(* Logix 5000 project; controller NSH_PLC2 vendor 1 type 14 code 167 rev 32.14; software revision 32.03; part 2 of 6 *)
(* tags used below, declared in another part *)
   AOI_MCC2_10A_ToPLC1 : E300ToMotor;
   AOI_MCC2_10C_ToPLC1 : E300ToMotor;
   AOI_MCC2_10E_ToPLC1 : E300ToMotor;
   AOI_MCC2_10G_ToPLC1 : E300ToMotor;
   AOI_MCC2_10J_ToPLC1 : E300ToMotor;
   AOI_MCC2_10L_ToPLC1 : E300ToMotor;
   AOI_MCC2_11A_ToPLC1 : E300ToMotor;
   AOI_MCC2_11C_ToPLC1 : E300ToMotor;
   AOI_MCC2_11E_ToPLC1 : E300ToMotor;
   AOI_MCC2_11G_ToPLC1 : E300ToMotor;
   AOI_MCC2_11J_ToPLC1 : E300ToMotor;
   AOI_MCC2_11L_ToPLC1 : E300ToMotor;
   AOI_MCC2_12A_ToPLC1 : E300ToMotor;
   AOI_MCC2_12C_ToPLC1 : E300ToMotor;
   AOI_MCC2_12E_ToPLC1 : E300ToMotor;
   AOI_MCC2_12G_ToPLC1 : E300ToMotor;
   AOI_MCC2_12J_ToPLC1 : E300ToMotor;
   AOI_MCC2_12L_ToPLC1 : E300ToMotor;
   AOI_MCC2_13A_ToPLC1 : E300ToMotor;
   AOI_MCC2_13C_ToPLC1 : E300ToMotor;
   AOI_MCC2_13E_ToPLC1 : E300ToMotor;
   AOI_MCC2_13G_ToPLC1 : E300ToMotor;
   AOI_MCC2_13J_ToPLC1 : E300ToMotor;
   AOI_MCC2_14A_ToPLC1 : E300ToMotor;
   AOI_MCC2_14C_ToPLC1 : E300ToMotor;
   AOI_MCC2_14E_ToPLC1 : E300ToMotor;
   AOI_MCC2_14G_ToPLC1 : E300ToMotor;
   AOI_MCC2_14J_ToPLC1 : E300ToMotor;
   AOI_MCC2_14L_ToPLC1 : E300ToMotor;
   AOI_MCC2_15A_ToPLC1 : E300ToMotor;
   AOI_MCC2_15C_ToPLC1 : E300ToMotor;
   AOI_MCC2_15E_ToPLC1 : E300ToMotor;
   AOI_MCC2_15G_ToPLC1 : E300ToMotor;
   AOI_MCC2_2A_ToPLC1 : PF525ToMotor;
   AOI_MCC2_2D_ToPLC1 : PF525ToMotor;
   AOI_MCC2_2G_ToPLC1 : PF525ToMotor;
   AOI_MCC2_2K_ToPLC1 : PF525ToMotor;
   AOI_MCC2_3A_ToPLC1 : E300ToMotor;
   AOI_MCC2_3C_ToPLC1 : E300ToMotor;
   AOI_MCC2_3E_ToPLC1 : E300ToMotor;
   AOI_MCC2_3G_ToPLC1 : E300ToMotor;
   AOI_MCC2_3J_ToPLC1 : E300ToMotor;
   AOI_MCC2_3L_ToPLC1 : E300ToMotor;
   AOI_MCC2_4A_ToPLC1 : E300ToMotor;
   AOI_MCC2_4C_ToPLC1 : E300ToMotor;
   AOI_MCC2_4E_ToPLC1 : E300ToMotor;
   AOI_MCC2_4G_ToPLC1 : E300ToMotor;
   AOI_MCC2_4J_ToPLC1 : E300ToMotor;
   AOI_MCC2_4L_ToPLC1 : E300ToMotor;
   AOI_MCC2_5A_ToPLC1 : E300ToMotor;
   AOI_MCC2_5C_ToPLC1 : E300ToMotor;
   AOI_MCC2_5E_ToPLC1 : E300ToMotor;
   AOI_MCC2_5G_ToPLC1 : E300ToMotor;
   AOI_MCC2_5J_ToPLC1 : E300ToMotor;
   AOI_MCC2_6A_ToPLC1 : E300ToMotor;
   AOI_MCC2_6C_ToPLC1 : E300ToMotor;
   AOI_MCC2_6E_ToPLC1 : E300ToMotor;
   AOI_MCC2_6G_ToPLC1 : E300ToMotor;
   AOI_MCC2_6J_ToPLC1 : E300ToMotor;
   AOI_MCC2_6L_ToPLC1 : E300ToMotor;
   AOI_MCC2_7A_ToPLC1 : E300ToMotor;
   AOI_MCC2_7D_ToPLC1 : E300ToMotor;
   AOI_MCC2_7G_ToPLC1 : E300ToMotor;
   AOI_MCC2_7K_ToPLC1 : E300ToMotor;
   AOI_MCC2_8B_ToPLC1 : E300ToMotor;
   AOI_MCC2_8D_ToPLC1 : E300ToMotor;
   AOI_MCC2_8F_ToPLC1 : E300ToMotor;
   AOI_MCC2_8H_ToPLC1 : E300ToMotor;
   AOI_MCC2_8K_ToPLC1 : E300ToMotor;
   AOI_MCC2_9D_ToPLC1 : E300ToMotor;
   AOI_MCC2_9F_ToPLC1 : E300ToMotor;
   AOI_MCC2_9H_ToPLC1 : PF525ToMotor;
   Const_4000_Hex : INT;   // Constant #16:4000, Entry Status Communicating
   GSV_EntryStatus : INT;   // GSV Entry Status, shold be #16:4000
   MCC2_10A_CommsOK : BOOL;   // Communications with AOP OK
   MCC2_10C_CommsOK : BOOL;   // Communications with AOP OK
   MCC2_10E_CommsOK : BOOL;   // Communications with AOP OK
   MCC2_10G_CommsOK : BOOL;   // Communications with AOP OK
   MCC2_10J_CommsOK : BOOL;   // Communications with AOP OK
   MCC2_10L_CommsOK : BOOL;   // Communications with AOP OK
   MCC2_11A_CommsOK : BOOL;   // Communications with AOP OK
   MCC2_11C_CommsOK : BOOL;   // Communications with AOP OK
   MCC2_11E_CommsOK : BOOL;   // Communications with AOP OK
   MCC2_11G_CommsOK : BOOL;   // Communications with AOP OK
   MCC2_11J_CommsOK : BOOL;   // Communications with AOP OK
   MCC2_11L_CommsOK : BOOL;   // Communications with AOP OK
   MCC2_12A_CommsOK : BOOL;   // Communications with AOP OK
   MCC2_12C_CommsOK : BOOL;   // Communications with AOP OK
   MCC2_12E_CommsOK : BOOL;   // Communications with AOP OK
   MCC2_12G_CommsOK : BOOL;   // Communications with AOP OK
   MCC2_12J_CommsOK : BOOL;   // Communications with AOP OK
   MCC2_12L_CommsOK : BOOL;   // Communications with AOP OK
   MCC2_13A_CommsOK : BOOL;   // Communications with AOP OK
   MCC2_13C_CommsOK : BOOL;   // Communications with AOP OK
   MCC2_13E_CommsOK : BOOL;   // Communications with AOP OK
   MCC2_13G_CommsOK : BOOL;   // Communications with AOP OK
   MCC2_13J_CommsOK : BOOL;   // Communications with AOP OK
   MCC2_14A_CommsOK : BOOL;   // Communications with AOP OK
   MCC2_14C_CommsOK : BOOL;   // Communications with AOP OK
   MCC2_14E_CommsOK : BOOL;   // Communications with AOP OK
   MCC2_14G_CommsOK : BOOL;   // Communications with AOP OK
   MCC2_14J_CommsOK : BOOL;   // Communications with AOP OK
   MCC2_14L_CommsOK : BOOL;   // Communications with AOP OK
   MCC2_15A_CommsOK : BOOL;   // Communications with AOP OK
   MCC2_15C_CommsOK : BOOL;   // Communications with AOP OK
   MCC2_15E_CommsOK : BOOL;   // Communications with AOP OK
   MCC2_15G_CommsOK : BOOL;   // Communications with AOP OK
   MCC2_2A_CommsOK : BOOL;   // Communications with AOP OK
   MCC2_2D_CommsOK : BOOL;   // Communications with AOP OK
   MCC2_2G_CommsOK : BOOL;   // Communications with AOP OK
   MCC2_2K_CommsOK : BOOL;   // Communications with AOP OK
   MCC2_3A_CommsOK : BOOL;   // Communications with AOP OK
   MCC2_3C_CommsOK : BOOL;   // Communications with AOP OK
   MCC2_3E_CommsOK : BOOL;   // Communications with AOP OK
   MCC2_3G_CommsOK : BOOL;   // Communications with AOP OK
   MCC2_3J_CommsOK : BOOL;   // Communications with AOP OK
   MCC2_3L_CommsOK : BOOL;   // Communications with AOP OK
   MCC2_4A_CommsOK : BOOL;   // Communications with AOP OK
   MCC2_4C_CommsOK : BOOL;   // Communications with AOP OK
   MCC2_4E_CommsOK : BOOL;   // Communications with AOP OK
   MCC2_4G_CommsOK : BOOL;   // Communications with AOP OK
   MCC2_4J_CommsOK : BOOL;   // Communications with AOP OK
   MCC2_4L_CommsOK : BOOL;   // Communications with AOP OK
   MCC2_5A_CommsOK : BOOL;   // Communications with AOP OK
   MCC2_5C_CommsOK : BOOL;   // Communications with AOP OK
   MCC2_5E_CommsOK : BOOL;   // Communications with AOP OK
   MCC2_5G_CommsOK : BOOL;   // Communications with AOP OK
   MCC2_5J_CommsOK : BOOL;   // Communications with AOP OK
   MCC2_6A_CommsOK : BOOL;   // Communications with AOP OK
   MCC2_6C_CommsOK : BOOL;   // Communications with AOP OK
   MCC2_6E_CommsOK : BOOL;   // Communications with AOP OK
   MCC2_6G_CommsOK : BOOL;   // Communications with AOP OK
   MCC2_6J_CommsOK : BOOL;   // Communications with AOP OK
   MCC2_6L_CommsOK1 : BOOL;   // Communications with AOP OK
   MCC2_7A_CommsOK : BOOL;   // Communications with AOP OK
   MCC2_7D_CommsOK : BOOL;   // Communications with AOP OK
   MCC2_7G_CommsOK : BOOL;   // Communications with AOP OK
   MCC2_7K_CommsOK : BOOL;   // Communications with AOP OK
   MCC2_8B_CommsOK : BOOL;   // Communications with AOP OK
   MCC2_8D_CommsOK : BOOL;   // Communications with AOP OK
   MCC2_8F_CommsOK : BOOL;   // Communications with AOP OK
   MCC2_8H_CommsOK : BOOL;   // Communications with AOP OK
   MCC2_8K_CommsOK : BOOL;   // Communications with AOP OK
   MCC2_9D_CommsOK : BOOL;   // Communications with AOP OK
   MCC2_9F_CommsOK : BOOL;   // Communications with AOP OK
   MCC2_9H_CommsOK : BOOL;   // Communications with AOP OK
   MotorsStatusTag : MotorsStatusUDT;   // Only Instance of UDT

PROGRAM MainProgram   (* main routine MainRoutine *)

ROUTINE AOP_ToPLC1   (* ladder *)
// Get Motor AOPs To AllMotorsToPLC1
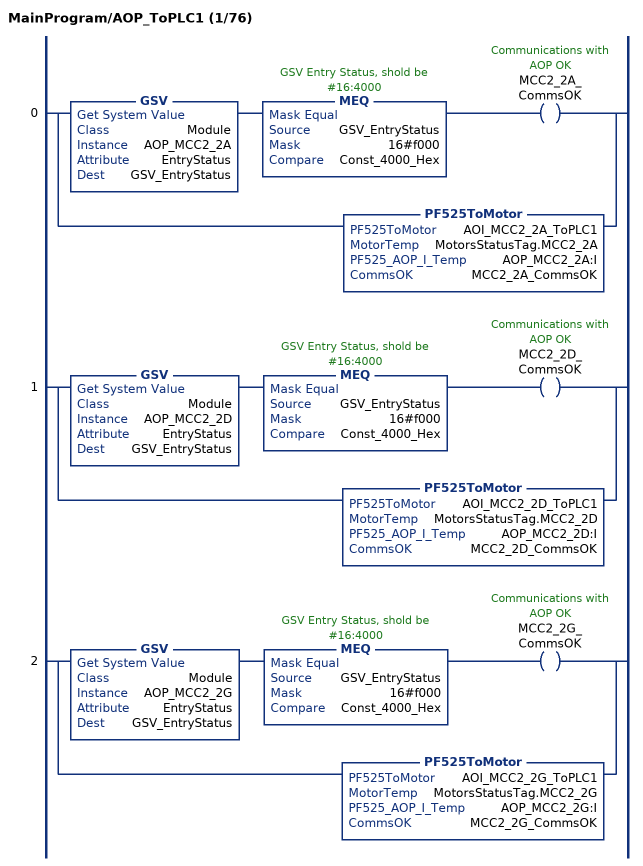
   0: [GSV(Module,AOP_MCC2_2A,EntryStatus,GSV_EntryStatus) MEQ(GSV_EntryStatus,16#f000,Const_4000_Hex) OTE(MCC2_2A_CommsOK) ,PF525ToMotor(AOI_MCC2_2A_ToPLC1,MotorsStatusTag.MCC2_2A,AOP_MCC2_2A:I,MCC2_2A_CommsOK) ];
   1: [GSV(Module,AOP_MCC2_2D,EntryStatus,GSV_EntryStatus) MEQ(GSV_EntryStatus,16#f000,Const_4000_Hex) OTE(MCC2_2D_CommsOK) ,PF525ToMotor(AOI_MCC2_2D_ToPLC1,MotorsStatusTag.MCC2_2D,AOP_MCC2_2D:I,MCC2_2D_CommsOK) ];
   2: [GSV(Module,AOP_MCC2_2G,EntryStatus,GSV_EntryStatus) MEQ(GSV_EntryStatus,16#f000,Const_4000_Hex) OTE(MCC2_2G_CommsOK) ,PF525ToMotor(AOI_MCC2_2G_ToPLC1,MotorsStatusTag.MCC2_2G,AOP_MCC2_2G:I,MCC2_2G_CommsOK) ];
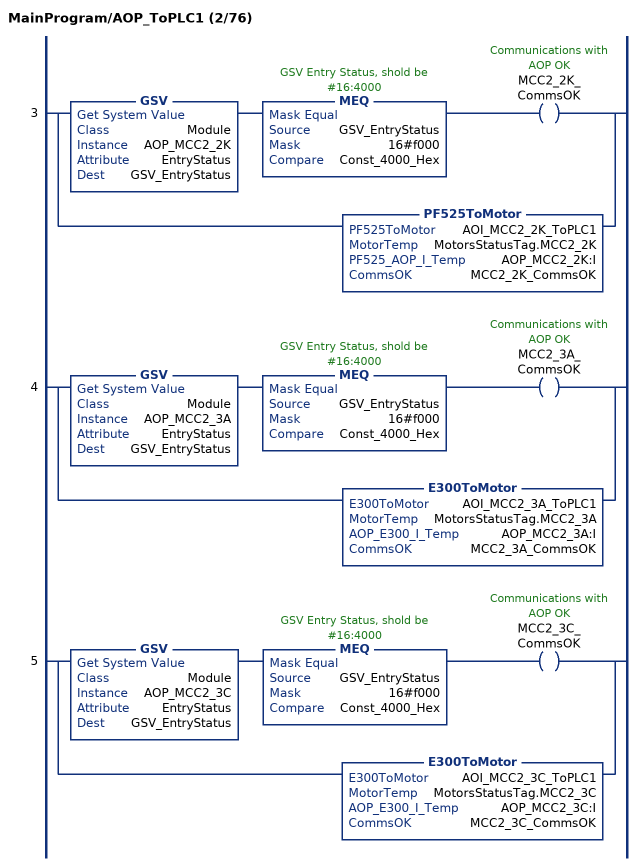
   3: [GSV(Module,AOP_MCC2_2K,EntryStatus,GSV_EntryStatus) MEQ(GSV_EntryStatus,16#f000,Const_4000_Hex) OTE(MCC2_2K_CommsOK) ,PF525ToMotor(AOI_MCC2_2K_ToPLC1,MotorsStatusTag.MCC2_2K,AOP_MCC2_2K:I,MCC2_2K_CommsOK) ];
   4: [GSV(Module,AOP_MCC2_3A,EntryStatus,GSV_EntryStatus) MEQ(GSV_EntryStatus,16#f000,Const_4000_Hex) OTE(MCC2_3A_CommsOK) ,E300ToMotor(AOI_MCC2_3A_ToPLC1,MotorsStatusTag.MCC2_3A,AOP_MCC2_3A:I,MCC2_3A_CommsOK) ];
   5: [GSV(Module,AOP_MCC2_3C,EntryStatus,GSV_EntryStatus) MEQ(GSV_EntryStatus,16#f000,Const_4000_Hex) OTE(MCC2_3C_CommsOK) ,E300ToMotor(AOI_MCC2_3C_ToPLC1,MotorsStatusTag.MCC2_3C,AOP_MCC2_3C:I,MCC2_3C_CommsOK) ];
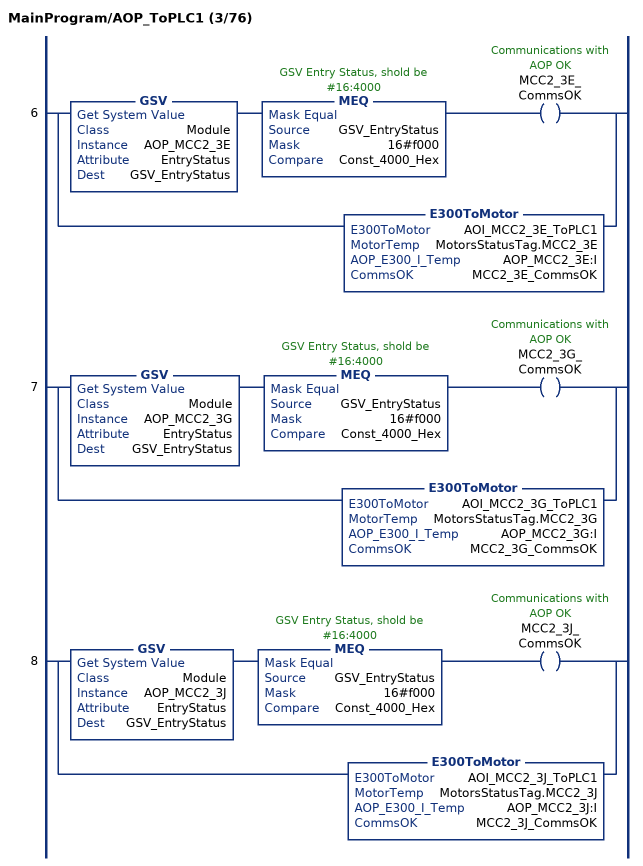
   6: [GSV(Module,AOP_MCC2_3E,EntryStatus,GSV_EntryStatus) MEQ(GSV_EntryStatus,16#f000,Const_4000_Hex) OTE(MCC2_3E_CommsOK) ,E300ToMotor(AOI_MCC2_3E_ToPLC1,MotorsStatusTag.MCC2_3E,AOP_MCC2_3E:I,MCC2_3E_CommsOK) ];
   7: [GSV(Module,AOP_MCC2_3G,EntryStatus,GSV_EntryStatus) MEQ(GSV_EntryStatus,16#f000,Const_4000_Hex) OTE(MCC2_3G_CommsOK) ,E300ToMotor(AOI_MCC2_3G_ToPLC1,MotorsStatusTag.MCC2_3G,AOP_MCC2_3G:I,MCC2_3G_CommsOK) ];
   8: [GSV(Module,AOP_MCC2_3J,EntryStatus,GSV_EntryStatus) MEQ(GSV_EntryStatus,16#f000,Const_4000_Hex) OTE(MCC2_3J_CommsOK) ,E300ToMotor(AOI_MCC2_3J_ToPLC1,MotorsStatusTag.MCC2_3J,AOP_MCC2_3J:I,MCC2_3J_CommsOK) ];
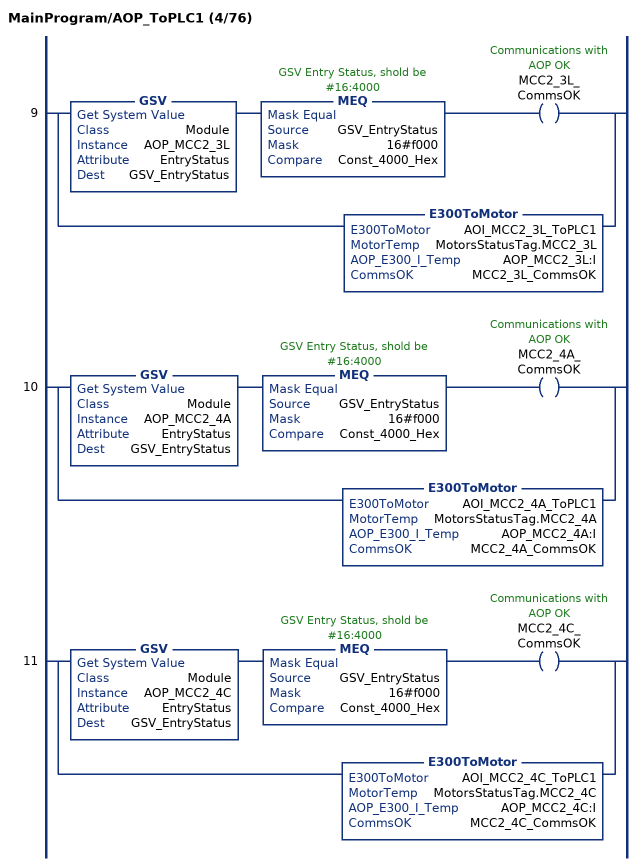
   9: [GSV(Module,AOP_MCC2_3L,EntryStatus,GSV_EntryStatus) MEQ(GSV_EntryStatus,16#f000,Const_4000_Hex) OTE(MCC2_3L_CommsOK) ,E300ToMotor(AOI_MCC2_3L_ToPLC1,MotorsStatusTag.MCC2_3L,AOP_MCC2_3L:I,MCC2_3L_CommsOK) ];
   10: [GSV(Module,AOP_MCC2_4A,EntryStatus,GSV_EntryStatus) MEQ(GSV_EntryStatus,16#f000,Const_4000_Hex) OTE(MCC2_4A_CommsOK) ,E300ToMotor(AOI_MCC2_4A_ToPLC1,MotorsStatusTag.MCC2_4A,AOP_MCC2_4A:I,MCC2_4A_CommsOK) ];
   11: [GSV(Module,AOP_MCC2_4C,EntryStatus,GSV_EntryStatus) MEQ(GSV_EntryStatus,16#f000,Const_4000_Hex) OTE(MCC2_4C_CommsOK) ,E300ToMotor(AOI_MCC2_4C_ToPLC1,MotorsStatusTag.MCC2_4C,AOP_MCC2_4C:I,MCC2_4C_CommsOK) ];
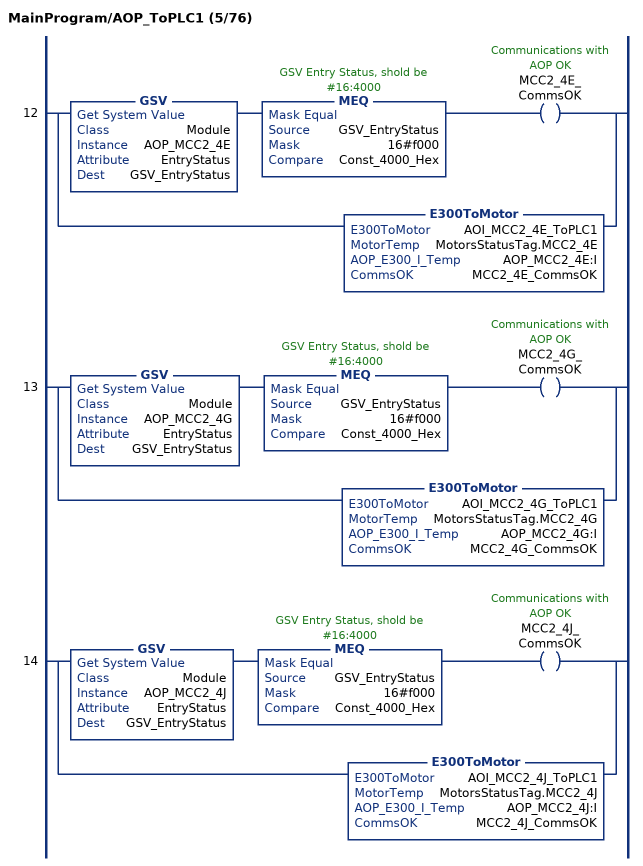
   12: [GSV(Module,AOP_MCC2_4E,EntryStatus,GSV_EntryStatus) MEQ(GSV_EntryStatus,16#f000,Const_4000_Hex) OTE(MCC2_4E_CommsOK) ,E300ToMotor(AOI_MCC2_4E_ToPLC1,MotorsStatusTag.MCC2_4E,AOP_MCC2_4E:I,MCC2_4E_CommsOK) ];
   13: [GSV(Module,AOP_MCC2_4G,EntryStatus,GSV_EntryStatus) MEQ(GSV_EntryStatus,16#f000,Const_4000_Hex) OTE(MCC2_4G_CommsOK) ,E300ToMotor(AOI_MCC2_4G_ToPLC1,MotorsStatusTag.MCC2_4G,AOP_MCC2_4G:I,MCC2_4G_CommsOK) ];
   14: [GSV(Module,AOP_MCC2_4J,EntryStatus,GSV_EntryStatus) MEQ(GSV_EntryStatus,16#f000,Const_4000_Hex) OTE(MCC2_4J_CommsOK) ,E300ToMotor(AOI_MCC2_4J_ToPLC1,MotorsStatusTag.MCC2_4J,AOP_MCC2_4J:I,MCC2_4J_CommsOK) ];
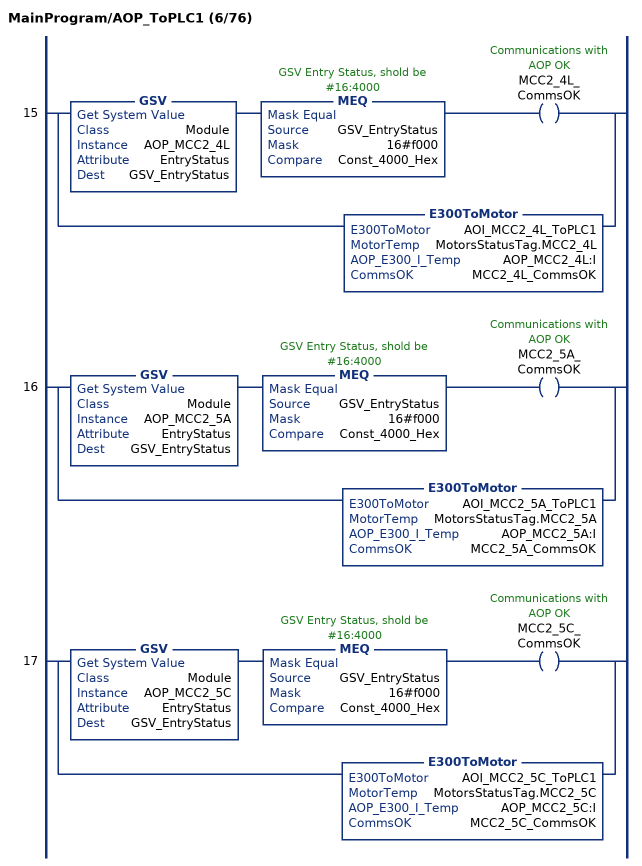
   15: [GSV(Module,AOP_MCC2_4L,EntryStatus,GSV_EntryStatus) MEQ(GSV_EntryStatus,16#f000,Const_4000_Hex) OTE(MCC2_4L_CommsOK) ,E300ToMotor(AOI_MCC2_4L_ToPLC1,MotorsStatusTag.MCC2_4L,AOP_MCC2_4L:I,MCC2_4L_CommsOK) ];
   16: [GSV(Module,AOP_MCC2_5A,EntryStatus,GSV_EntryStatus) MEQ(GSV_EntryStatus,16#f000,Const_4000_Hex) OTE(MCC2_5A_CommsOK) ,E300ToMotor(AOI_MCC2_5A_ToPLC1,MotorsStatusTag.MCC2_5A,AOP_MCC2_5A:I,MCC2_5A_CommsOK) ];
   17: [GSV(Module,AOP_MCC2_5C,EntryStatus,GSV_EntryStatus) MEQ(GSV_EntryStatus,16#f000,Const_4000_Hex) OTE(MCC2_5C_CommsOK) ,E300ToMotor(AOI_MCC2_5C_ToPLC1,MotorsStatusTag.MCC2_5C,AOP_MCC2_5C:I,MCC2_5C_CommsOK) ];
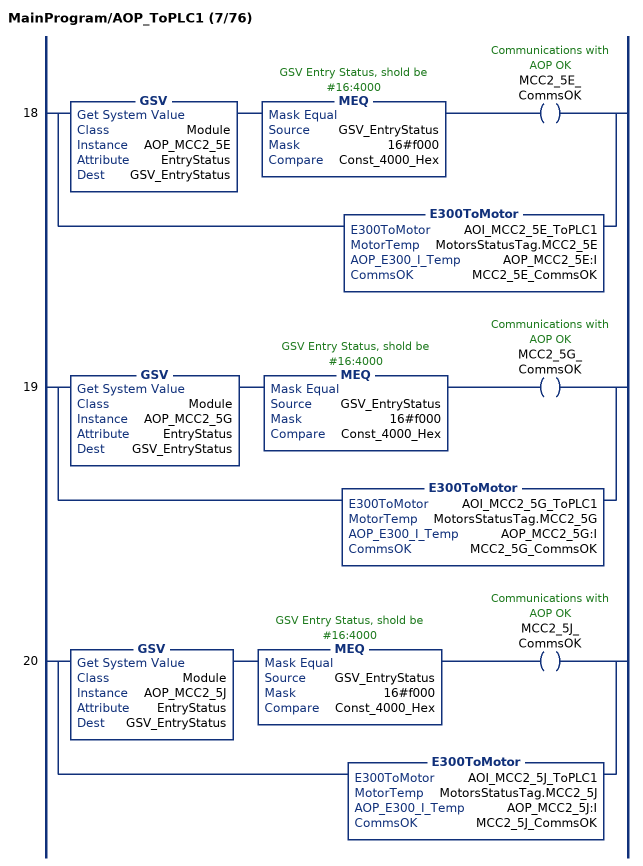
   18: [GSV(Module,AOP_MCC2_5E,EntryStatus,GSV_EntryStatus) MEQ(GSV_EntryStatus,16#f000,Const_4000_Hex) OTE(MCC2_5E_CommsOK) ,E300ToMotor(AOI_MCC2_5E_ToPLC1,MotorsStatusTag.MCC2_5E,AOP_MCC2_5E:I,MCC2_5E_CommsOK) ];
   19: [GSV(Module,AOP_MCC2_5G,EntryStatus,GSV_EntryStatus) MEQ(GSV_EntryStatus,16#f000,Const_4000_Hex) OTE(MCC2_5G_CommsOK) ,E300ToMotor(AOI_MCC2_5G_ToPLC1,MotorsStatusTag.MCC2_5G,AOP_MCC2_5G:I,MCC2_5G_CommsOK) ];
   20: [GSV(Module,AOP_MCC2_5J,EntryStatus,GSV_EntryStatus) MEQ(GSV_EntryStatus,16#f000,Const_4000_Hex) OTE(MCC2_5J_CommsOK) ,E300ToMotor(AOI_MCC2_5J_ToPLC1,MotorsStatusTag.MCC2_5J,AOP_MCC2_5J:I,MCC2_5J_CommsOK) ];
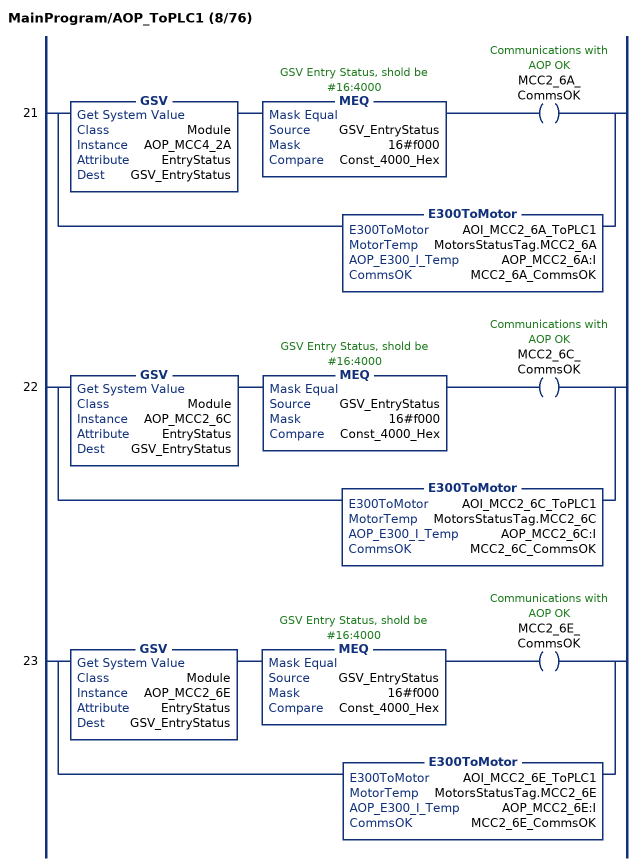
   21: [GSV(Module,AOP_MCC4_2A,EntryStatus,GSV_EntryStatus) MEQ(GSV_EntryStatus,16#f000,Const_4000_Hex) OTE(MCC2_6A_CommsOK) ,E300ToMotor(AOI_MCC2_6A_ToPLC1,MotorsStatusTag.MCC2_6A,AOP_MCC2_6A:I,MCC2_6A_CommsOK) ];
   22: [GSV(Module,AOP_MCC2_6C,EntryStatus,GSV_EntryStatus) MEQ(GSV_EntryStatus,16#f000,Const_4000_Hex) OTE(MCC2_6C_CommsOK) ,E300ToMotor(AOI_MCC2_6C_ToPLC1,MotorsStatusTag.MCC2_6C,AOP_MCC2_6C:I,MCC2_6C_CommsOK) ];
   23: [GSV(Module,AOP_MCC2_6E,EntryStatus,GSV_EntryStatus) MEQ(GSV_EntryStatus,16#f000,Const_4000_Hex) OTE(MCC2_6E_CommsOK) ,E300ToMotor(AOI_MCC2_6E_ToPLC1,MotorsStatusTag.MCC2_6E,AOP_MCC2_6E:I,MCC2_6E_CommsOK) ];
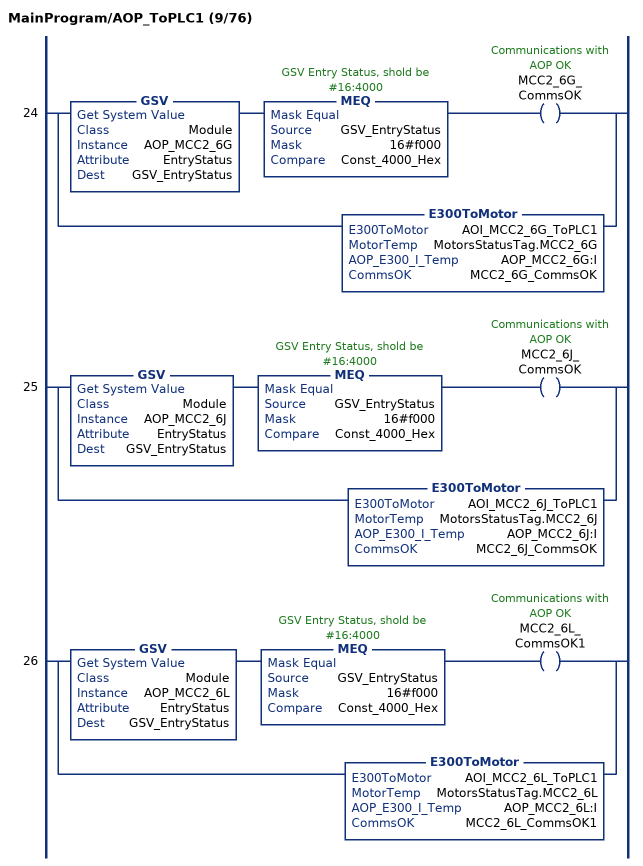
   24: [GSV(Module,AOP_MCC2_6G,EntryStatus,GSV_EntryStatus) MEQ(GSV_EntryStatus,16#f000,Const_4000_Hex) OTE(MCC2_6G_CommsOK) ,E300ToMotor(AOI_MCC2_6G_ToPLC1,MotorsStatusTag.MCC2_6G,AOP_MCC2_6G:I,MCC2_6G_CommsOK) ];
   25: [GSV(Module,AOP_MCC2_6J,EntryStatus,GSV_EntryStatus) MEQ(GSV_EntryStatus,16#f000,Const_4000_Hex) OTE(MCC2_6J_CommsOK) ,E300ToMotor(AOI_MCC2_6J_ToPLC1,MotorsStatusTag.MCC2_6J,AOP_MCC2_6J:I,MCC2_6J_CommsOK) ];
   26: [GSV(Module,AOP_MCC2_6L,EntryStatus,GSV_EntryStatus) MEQ(GSV_EntryStatus,16#f000,Const_4000_Hex) OTE(MCC2_6L_CommsOK1) ,E300ToMotor(AOI_MCC2_6L_ToPLC1,MotorsStatusTag.MCC2_6L,AOP_MCC2_6L:I,MCC2_6L_CommsOK1) ];
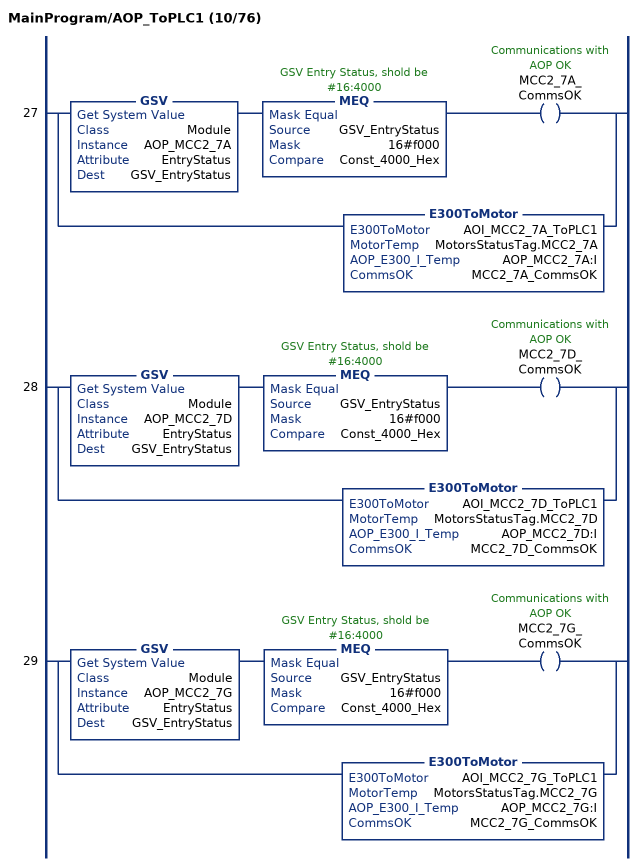
   27: [GSV(Module,AOP_MCC2_7A,EntryStatus,GSV_EntryStatus) MEQ(GSV_EntryStatus,16#f000,Const_4000_Hex) OTE(MCC2_7A_CommsOK) ,E300ToMotor(AOI_MCC2_7A_ToPLC1,MotorsStatusTag.MCC2_7A,AOP_MCC2_7A:I,MCC2_7A_CommsOK) ];
   28: [GSV(Module,AOP_MCC2_7D,EntryStatus,GSV_EntryStatus) MEQ(GSV_EntryStatus,16#f000,Const_4000_Hex) OTE(MCC2_7D_CommsOK) ,E300ToMotor(AOI_MCC2_7D_ToPLC1,MotorsStatusTag.MCC2_7D,AOP_MCC2_7D:I,MCC2_7D_CommsOK) ];
   29: [GSV(Module,AOP_MCC2_7G,EntryStatus,GSV_EntryStatus) MEQ(GSV_EntryStatus,16#f000,Const_4000_Hex) OTE(MCC2_7G_CommsOK) ,E300ToMotor(AOI_MCC2_7G_ToPLC1,MotorsStatusTag.MCC2_7G,AOP_MCC2_7G:I,MCC2_7G_CommsOK) ];
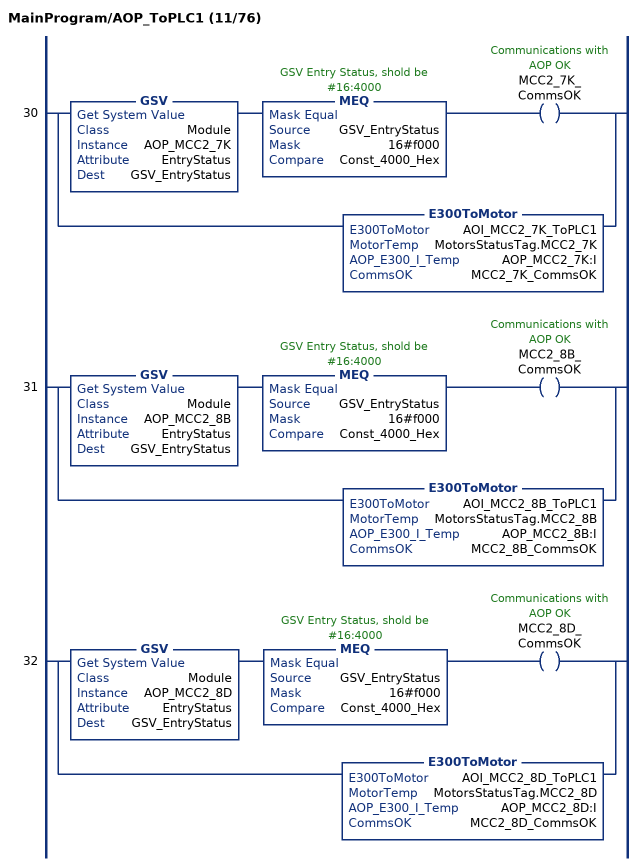
   30: [GSV(Module,AOP_MCC2_7K,EntryStatus,GSV_EntryStatus) MEQ(GSV_EntryStatus,16#f000,Const_4000_Hex) OTE(MCC2_7K_CommsOK) ,E300ToMotor(AOI_MCC2_7K_ToPLC1,MotorsStatusTag.MCC2_7K,AOP_MCC2_7K:I,MCC2_7K_CommsOK) ];
   31: [GSV(Module,AOP_MCC2_8B,EntryStatus,GSV_EntryStatus) MEQ(GSV_EntryStatus,16#f000,Const_4000_Hex) OTE(MCC2_8B_CommsOK) ,E300ToMotor(AOI_MCC2_8B_ToPLC1,MotorsStatusTag.MCC2_8B,AOP_MCC2_8B:I,MCC2_8B_CommsOK) ];
   32: [GSV(Module,AOP_MCC2_8D,EntryStatus,GSV_EntryStatus) MEQ(GSV_EntryStatus,16#f000,Const_4000_Hex) OTE(MCC2_8D_CommsOK) ,E300ToMotor(AOI_MCC2_8D_ToPLC1,MotorsStatusTag.MCC2_8D,AOP_MCC2_8D:I,MCC2_8D_CommsOK) ];
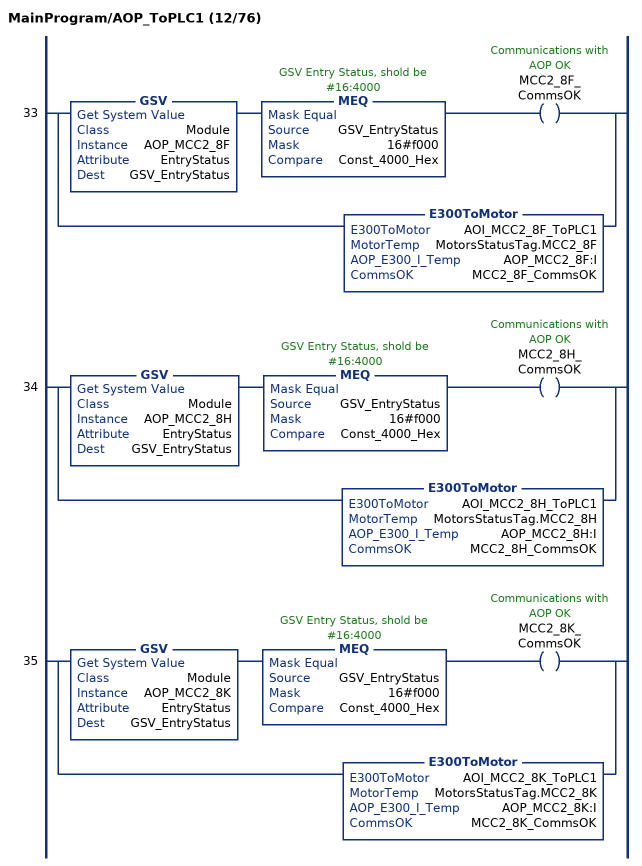
   33: [GSV(Module,AOP_MCC2_8F,EntryStatus,GSV_EntryStatus) MEQ(GSV_EntryStatus,16#f000,Const_4000_Hex) OTE(MCC2_8F_CommsOK) ,E300ToMotor(AOI_MCC2_8F_ToPLC1,MotorsStatusTag.MCC2_8F,AOP_MCC2_8F:I,MCC2_8F_CommsOK) ];
   34: [GSV(Module,AOP_MCC2_8H,EntryStatus,GSV_EntryStatus) MEQ(GSV_EntryStatus,16#f000,Const_4000_Hex) OTE(MCC2_8H_CommsOK) ,E300ToMotor(AOI_MCC2_8H_ToPLC1,MotorsStatusTag.MCC2_8H,AOP_MCC2_8H:I,MCC2_8H_CommsOK) ];
   35: [GSV(Module,AOP_MCC2_8K,EntryStatus,GSV_EntryStatus) MEQ(GSV_EntryStatus,16#f000,Const_4000_Hex) OTE(MCC2_8K_CommsOK) ,E300ToMotor(AOI_MCC2_8K_ToPLC1,MotorsStatusTag.MCC2_8K,AOP_MCC2_8K:I,MCC2_8K_CommsOK) ];
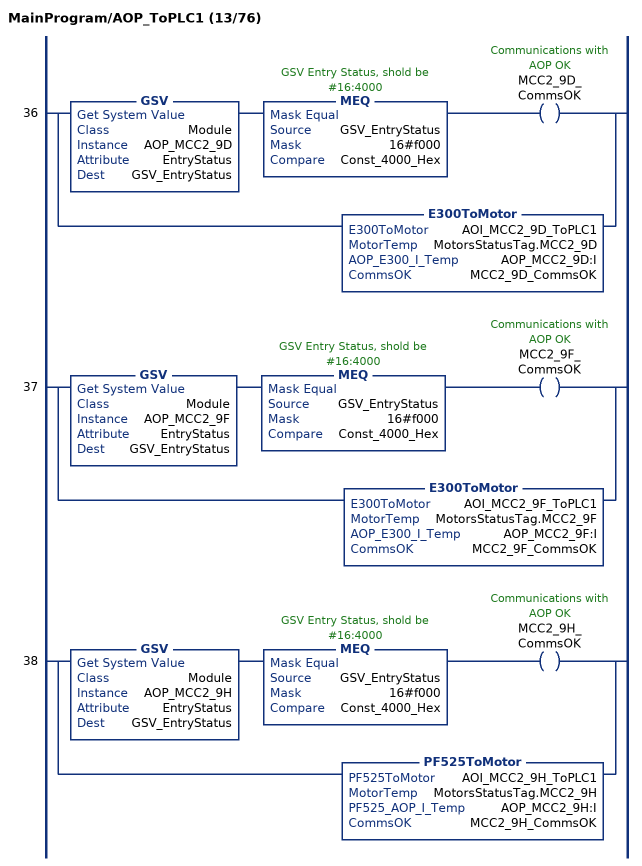
   36: [GSV(Module,AOP_MCC2_9D,EntryStatus,GSV_EntryStatus) MEQ(GSV_EntryStatus,16#f000,Const_4000_Hex) OTE(MCC2_9D_CommsOK) ,E300ToMotor(AOI_MCC2_9D_ToPLC1,MotorsStatusTag.MCC2_9D,AOP_MCC2_9D:I,MCC2_9D_CommsOK) ];
   37: [GSV(Module,AOP_MCC2_9F,EntryStatus,GSV_EntryStatus) MEQ(GSV_EntryStatus,16#f000,Const_4000_Hex) OTE(MCC2_9F_CommsOK) ,E300ToMotor(AOI_MCC2_9F_ToPLC1,MotorsStatusTag.MCC2_9F,AOP_MCC2_9F:I,MCC2_9F_CommsOK) ];
   38: [GSV(Module,AOP_MCC2_9H,EntryStatus,GSV_EntryStatus) MEQ(GSV_EntryStatus,16#f000,Const_4000_Hex) OTE(MCC2_9H_CommsOK) ,PF525ToMotor(AOI_MCC2_9H_ToPLC1,MotorsStatusTag.MCC2_9H,AOP_MCC2_9H:I,MCC2_9H_CommsOK) ];
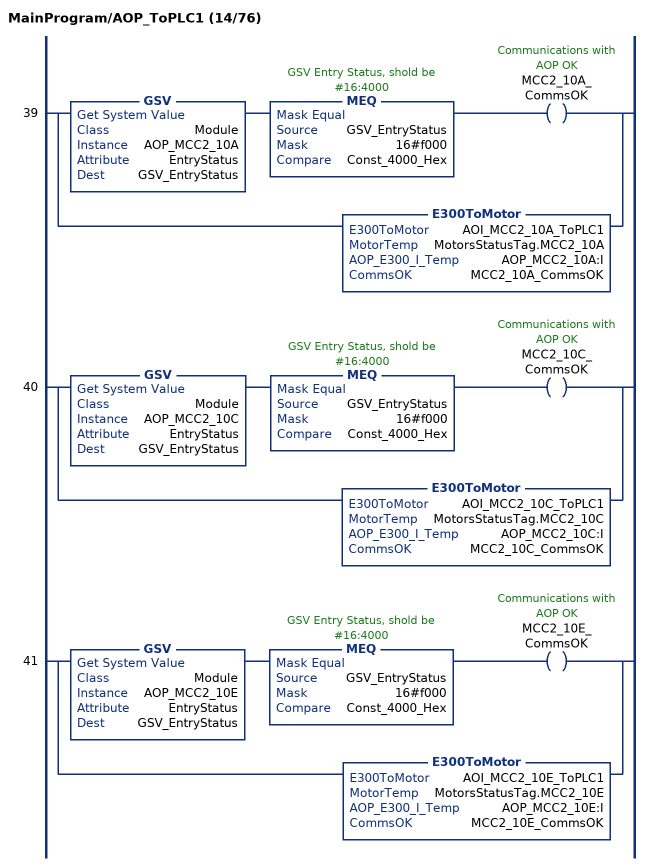
   39: [GSV(Module,AOP_MCC2_10A,EntryStatus,GSV_EntryStatus) MEQ(GSV_EntryStatus,16#f000,Const_4000_Hex) OTE(MCC2_10A_CommsOK) ,E300ToMotor(AOI_MCC2_10A_ToPLC1,MotorsStatusTag.MCC2_10A,AOP_MCC2_10A:I,MCC2_10A_CommsOK) ];
   40: [GSV(Module,AOP_MCC2_10C,EntryStatus,GSV_EntryStatus) MEQ(GSV_EntryStatus,16#f000,Const_4000_Hex) OTE(MCC2_10C_CommsOK) ,E300ToMotor(AOI_MCC2_10C_ToPLC1,MotorsStatusTag.MCC2_10C,AOP_MCC2_10C:I,MCC2_10C_CommsOK) ];
   41: [GSV(Module,AOP_MCC2_10E,EntryStatus,GSV_EntryStatus) MEQ(GSV_EntryStatus,16#f000,Const_4000_Hex) OTE(MCC2_10E_CommsOK) ,E300ToMotor(AOI_MCC2_10E_ToPLC1,MotorsStatusTag.MCC2_10E,AOP_MCC2_10E:I,MCC2_10E_CommsOK) ];
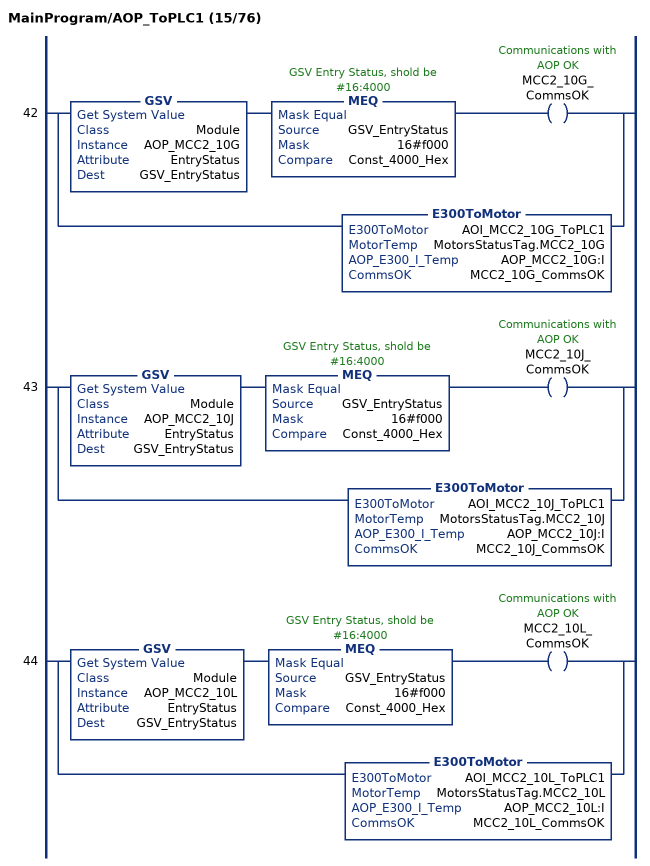
   42: [GSV(Module,AOP_MCC2_10G,EntryStatus,GSV_EntryStatus) MEQ(GSV_EntryStatus,16#f000,Const_4000_Hex) OTE(MCC2_10G_CommsOK) ,E300ToMotor(AOI_MCC2_10G_ToPLC1,MotorsStatusTag.MCC2_10G,AOP_MCC2_10G:I,MCC2_10G_CommsOK) ];
   43: [GSV(Module,AOP_MCC2_10J,EntryStatus,GSV_EntryStatus) MEQ(GSV_EntryStatus,16#f000,Const_4000_Hex) OTE(MCC2_10J_CommsOK) ,E300ToMotor(AOI_MCC2_10J_ToPLC1,MotorsStatusTag.MCC2_10J,AOP_MCC2_10J:I,MCC2_10J_CommsOK) ];
   44: [GSV(Module,AOP_MCC2_10L,EntryStatus,GSV_EntryStatus) MEQ(GSV_EntryStatus,16#f000,Const_4000_Hex) OTE(MCC2_10L_CommsOK) ,E300ToMotor(AOI_MCC2_10L_ToPLC1,MotorsStatusTag.MCC2_10L,AOP_MCC2_10L:I,MCC2_10L_CommsOK) ];
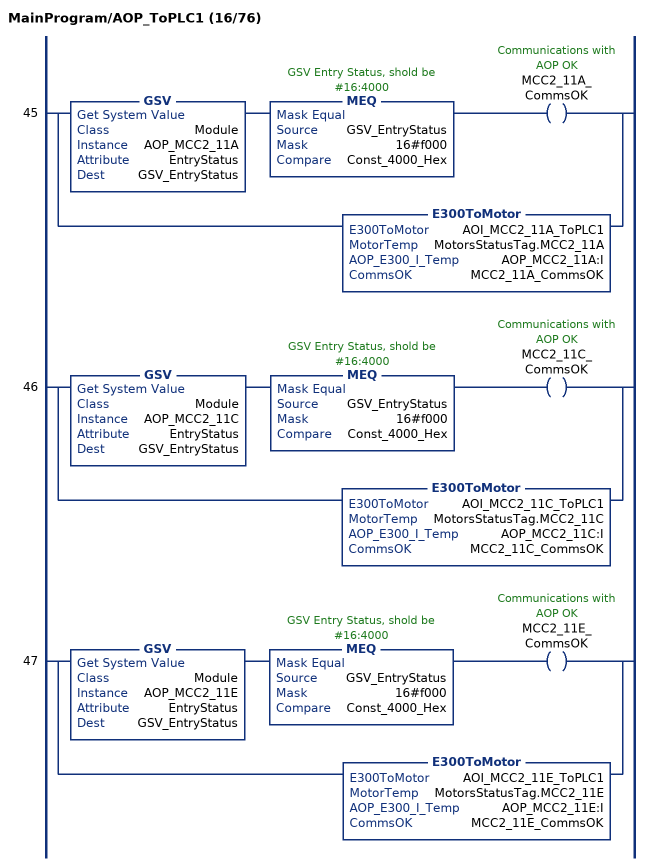
   45: [GSV(Module,AOP_MCC2_11A,EntryStatus,GSV_EntryStatus) MEQ(GSV_EntryStatus,16#f000,Const_4000_Hex) OTE(MCC2_11A_CommsOK) ,E300ToMotor(AOI_MCC2_11A_ToPLC1,MotorsStatusTag.MCC2_11A,AOP_MCC2_11A:I,MCC2_11A_CommsOK) ];
   46: [GSV(Module,AOP_MCC2_11C,EntryStatus,GSV_EntryStatus) MEQ(GSV_EntryStatus,16#f000,Const_4000_Hex) OTE(MCC2_11C_CommsOK) ,E300ToMotor(AOI_MCC2_11C_ToPLC1,MotorsStatusTag.MCC2_11C,AOP_MCC2_11C:I,MCC2_11C_CommsOK) ];
   47: [GSV(Module,AOP_MCC2_11E,EntryStatus,GSV_EntryStatus) MEQ(GSV_EntryStatus,16#f000,Const_4000_Hex) OTE(MCC2_11E_CommsOK) ,E300ToMotor(AOI_MCC2_11E_ToPLC1,MotorsStatusTag.MCC2_11E,AOP_MCC2_11E:I,MCC2_11E_CommsOK) ];
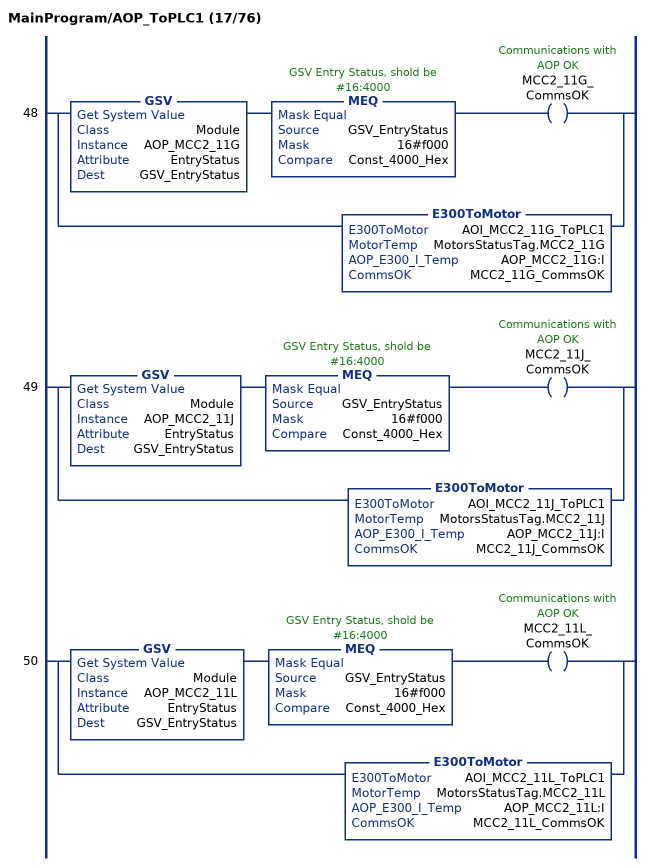
   48: [GSV(Module,AOP_MCC2_11G,EntryStatus,GSV_EntryStatus) MEQ(GSV_EntryStatus,16#f000,Const_4000_Hex) OTE(MCC2_11G_CommsOK) ,E300ToMotor(AOI_MCC2_11G_ToPLC1,MotorsStatusTag.MCC2_11G,AOP_MCC2_11G:I,MCC2_11G_CommsOK) ];
   49: [GSV(Module,AOP_MCC2_11J,EntryStatus,GSV_EntryStatus) MEQ(GSV_EntryStatus,16#f000,Const_4000_Hex) OTE(MCC2_11J_CommsOK) ,E300ToMotor(AOI_MCC2_11J_ToPLC1,MotorsStatusTag.MCC2_11J,AOP_MCC2_11J:I,MCC2_11J_CommsOK) ];
   50: [GSV(Module,AOP_MCC2_11L,EntryStatus,GSV_EntryStatus) MEQ(GSV_EntryStatus,16#f000,Const_4000_Hex) OTE(MCC2_11L_CommsOK) ,E300ToMotor(AOI_MCC2_11L_ToPLC1,MotorsStatusTag.MCC2_11L,AOP_MCC2_11L:I,MCC2_11L_CommsOK) ];
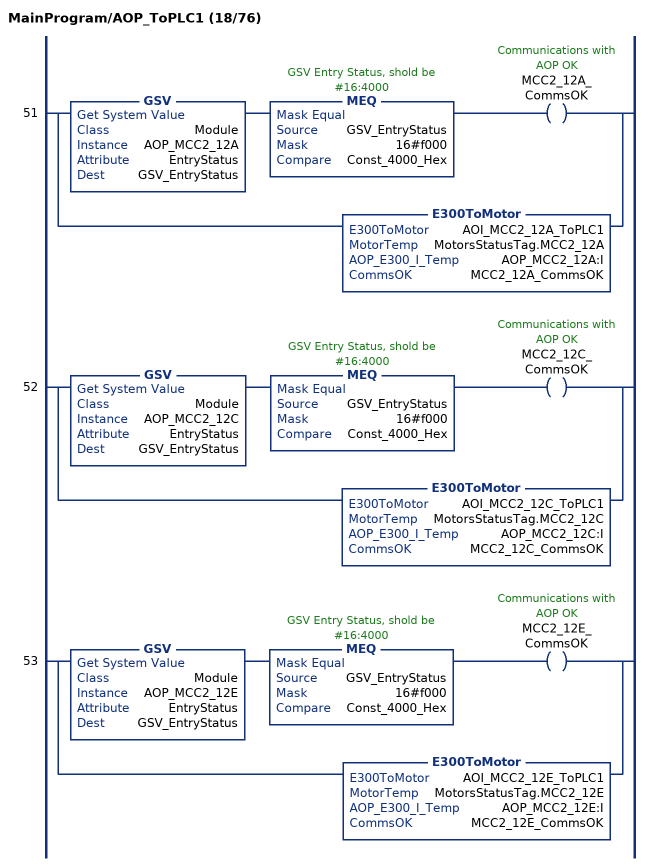
   51: [GSV(Module,AOP_MCC2_12A,EntryStatus,GSV_EntryStatus) MEQ(GSV_EntryStatus,16#f000,Const_4000_Hex) OTE(MCC2_12A_CommsOK) ,E300ToMotor(AOI_MCC2_12A_ToPLC1,MotorsStatusTag.MCC2_12A,AOP_MCC2_12A:I,MCC2_12A_CommsOK) ];
   52: [GSV(Module,AOP_MCC2_12C,EntryStatus,GSV_EntryStatus) MEQ(GSV_EntryStatus,16#f000,Const_4000_Hex) OTE(MCC2_12C_CommsOK) ,E300ToMotor(AOI_MCC2_12C_ToPLC1,MotorsStatusTag.MCC2_12C,AOP_MCC2_12C:I,MCC2_12C_CommsOK) ];
   53: [GSV(Module,AOP_MCC2_12E,EntryStatus,GSV_EntryStatus) MEQ(GSV_EntryStatus,16#f000,Const_4000_Hex) OTE(MCC2_12E_CommsOK) ,E300ToMotor(AOI_MCC2_12E_ToPLC1,MotorsStatusTag.MCC2_12E,AOP_MCC2_12E:I,MCC2_12E_CommsOK) ];
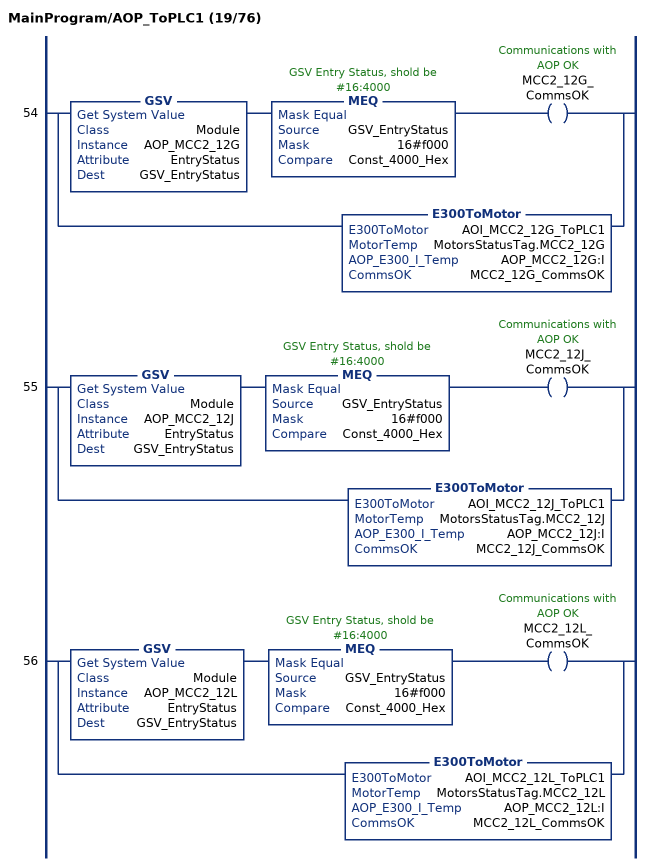
   54: [GSV(Module,AOP_MCC2_12G,EntryStatus,GSV_EntryStatus) MEQ(GSV_EntryStatus,16#f000,Const_4000_Hex) OTE(MCC2_12G_CommsOK) ,E300ToMotor(AOI_MCC2_12G_ToPLC1,MotorsStatusTag.MCC2_12G,AOP_MCC2_12G:I,MCC2_12G_CommsOK) ];
   55: [GSV(Module,AOP_MCC2_12J,EntryStatus,GSV_EntryStatus) MEQ(GSV_EntryStatus,16#f000,Const_4000_Hex) OTE(MCC2_12J_CommsOK) ,E300ToMotor(AOI_MCC2_12J_ToPLC1,MotorsStatusTag.MCC2_12J,AOP_MCC2_12J:I,MCC2_12J_CommsOK) ];
   56: [GSV(Module,AOP_MCC2_12L,EntryStatus,GSV_EntryStatus) MEQ(GSV_EntryStatus,16#f000,Const_4000_Hex) OTE(MCC2_12L_CommsOK) ,E300ToMotor(AOI_MCC2_12L_ToPLC1,MotorsStatusTag.MCC2_12L,AOP_MCC2_12L:I,MCC2_12L_CommsOK) ];
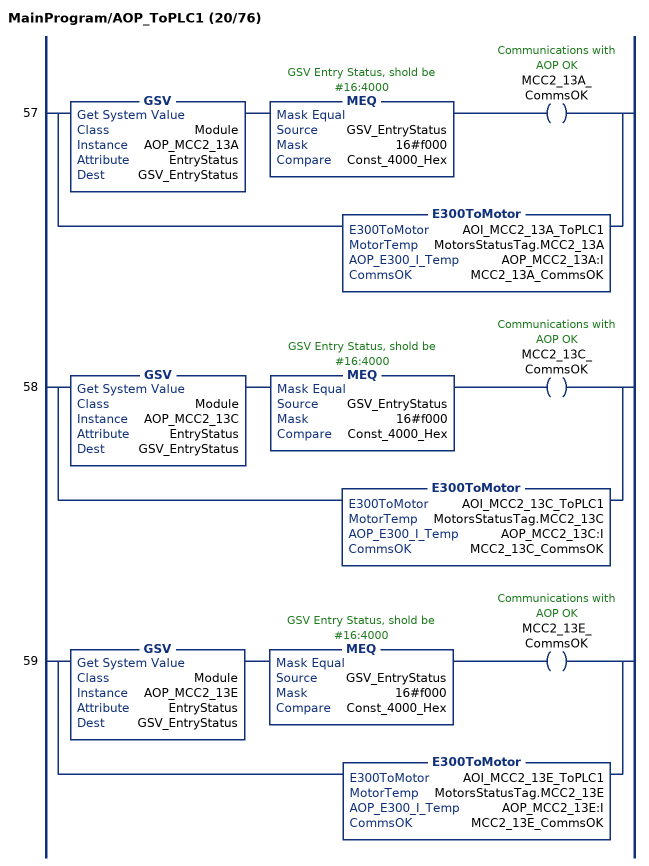
   57: [GSV(Module,AOP_MCC2_13A,EntryStatus,GSV_EntryStatus) MEQ(GSV_EntryStatus,16#f000,Const_4000_Hex) OTE(MCC2_13A_CommsOK) ,E300ToMotor(AOI_MCC2_13A_ToPLC1,MotorsStatusTag.MCC2_13A,AOP_MCC2_13A:I,MCC2_13A_CommsOK) ];
   58: [GSV(Module,AOP_MCC2_13C,EntryStatus,GSV_EntryStatus) MEQ(GSV_EntryStatus,16#f000,Const_4000_Hex) OTE(MCC2_13C_CommsOK) ,E300ToMotor(AOI_MCC2_13C_ToPLC1,MotorsStatusTag.MCC2_13C,AOP_MCC2_13C:I,MCC2_13C_CommsOK) ];
   59: [GSV(Module,AOP_MCC2_13E,EntryStatus,GSV_EntryStatus) MEQ(GSV_EntryStatus,16#f000,Const_4000_Hex) OTE(MCC2_13E_CommsOK) ,E300ToMotor(AOI_MCC2_13E_ToPLC1,MotorsStatusTag.MCC2_13E,AOP_MCC2_13E:I,MCC2_13E_CommsOK) ];
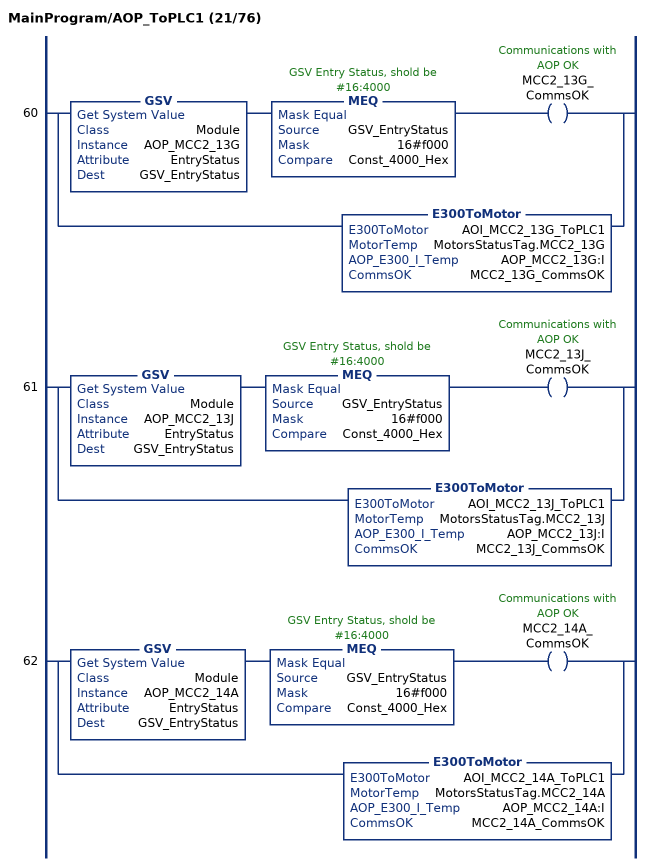
   60: [GSV(Module,AOP_MCC2_13G,EntryStatus,GSV_EntryStatus) MEQ(GSV_EntryStatus,16#f000,Const_4000_Hex) OTE(MCC2_13G_CommsOK) ,E300ToMotor(AOI_MCC2_13G_ToPLC1,MotorsStatusTag.MCC2_13G,AOP_MCC2_13G:I,MCC2_13G_CommsOK) ];
   61: [GSV(Module,AOP_MCC2_13J,EntryStatus,GSV_EntryStatus) MEQ(GSV_EntryStatus,16#f000,Const_4000_Hex) OTE(MCC2_13J_CommsOK) ,E300ToMotor(AOI_MCC2_13J_ToPLC1,MotorsStatusTag.MCC2_13J,AOP_MCC2_13J:I,MCC2_13J_CommsOK) ];
   62: [GSV(Module,AOP_MCC2_14A,EntryStatus,GSV_EntryStatus) MEQ(GSV_EntryStatus,16#f000,Const_4000_Hex) OTE(MCC2_14A_CommsOK) ,E300ToMotor(AOI_MCC2_14A_ToPLC1,MotorsStatusTag.MCC2_14A,AOP_MCC2_14A:I,MCC2_14A_CommsOK) ];
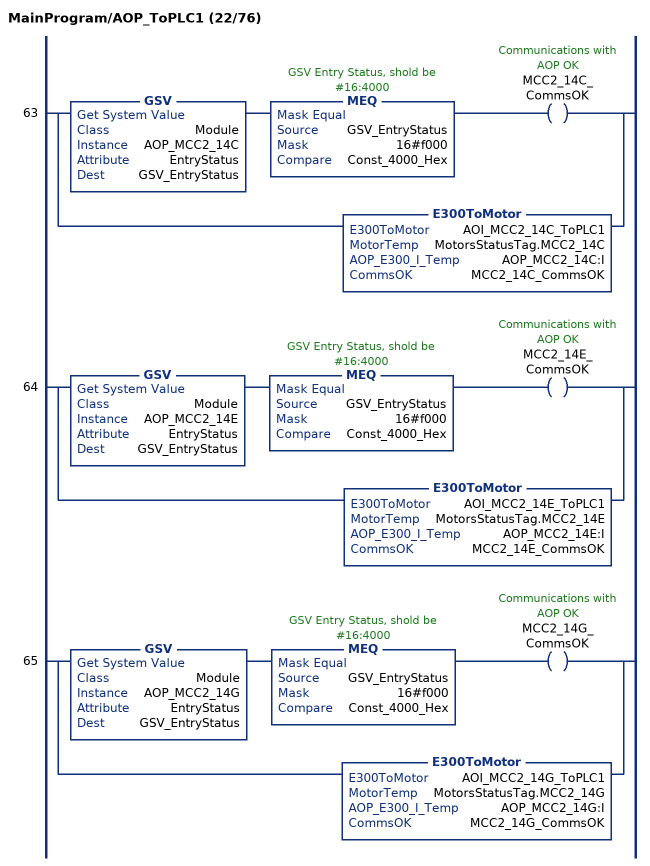
   63: [GSV(Module,AOP_MCC2_14C,EntryStatus,GSV_EntryStatus) MEQ(GSV_EntryStatus,16#f000,Const_4000_Hex) OTE(MCC2_14C_CommsOK) ,E300ToMotor(AOI_MCC2_14C_ToPLC1,MotorsStatusTag.MCC2_14C,AOP_MCC2_14C:I,MCC2_14C_CommsOK) ];
   64: [GSV(Module,AOP_MCC2_14E,EntryStatus,GSV_EntryStatus) MEQ(GSV_EntryStatus,16#f000,Const_4000_Hex) OTE(MCC2_14E_CommsOK) ,E300ToMotor(AOI_MCC2_14E_ToPLC1,MotorsStatusTag.MCC2_14E,AOP_MCC2_14E:I,MCC2_14E_CommsOK) ];
   65: [GSV(Module,AOP_MCC2_14G,EntryStatus,GSV_EntryStatus) MEQ(GSV_EntryStatus,16#f000,Const_4000_Hex) OTE(MCC2_14G_CommsOK) ,E300ToMotor(AOI_MCC2_14G_ToPLC1,MotorsStatusTag.MCC2_14G,AOP_MCC2_14G:I,MCC2_14G_CommsOK) ];
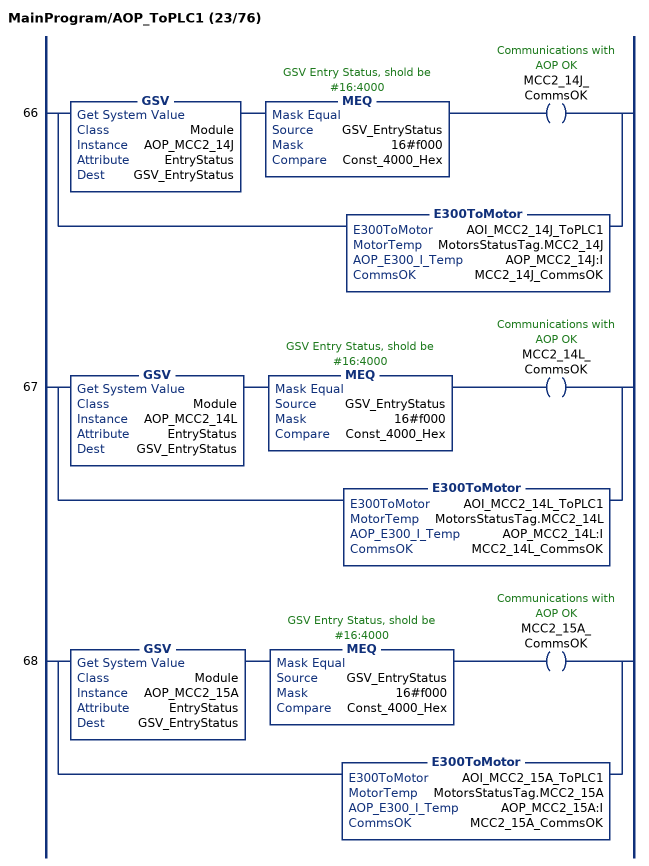
   66: [GSV(Module,AOP_MCC2_14J,EntryStatus,GSV_EntryStatus) MEQ(GSV_EntryStatus,16#f000,Const_4000_Hex) OTE(MCC2_14J_CommsOK) ,E300ToMotor(AOI_MCC2_14J_ToPLC1,MotorsStatusTag.MCC2_14J,AOP_MCC2_14J:I,MCC2_14J_CommsOK) ];
   67: [GSV(Module,AOP_MCC2_14L,EntryStatus,GSV_EntryStatus) MEQ(GSV_EntryStatus,16#f000,Const_4000_Hex) OTE(MCC2_14L_CommsOK) ,E300ToMotor(AOI_MCC2_14L_ToPLC1,MotorsStatusTag.MCC2_14L,AOP_MCC2_14L:I,MCC2_14L_CommsOK) ];
   68: [GSV(Module,AOP_MCC2_15A,EntryStatus,GSV_EntryStatus) MEQ(GSV_EntryStatus,16#f000,Const_4000_Hex) OTE(MCC2_15A_CommsOK) ,E300ToMotor(AOI_MCC2_15A_ToPLC1,MotorsStatusTag.MCC2_15A,AOP_MCC2_15A:I,MCC2_15A_CommsOK) ];
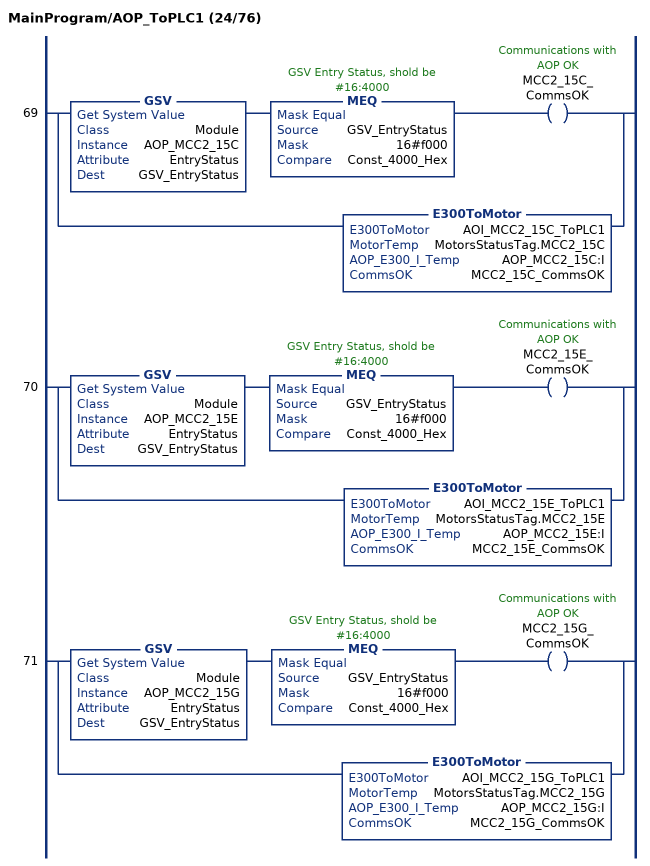
   69: [GSV(Module,AOP_MCC2_15C,EntryStatus,GSV_EntryStatus) MEQ(GSV_EntryStatus,16#f000,Const_4000_Hex) OTE(MCC2_15C_CommsOK) ,E300ToMotor(AOI_MCC2_15C_ToPLC1,MotorsStatusTag.MCC2_15C,AOP_MCC2_15C:I,MCC2_15C_CommsOK) ];
   70: [GSV(Module,AOP_MCC2_15E,EntryStatus,GSV_EntryStatus) MEQ(GSV_EntryStatus,16#f000,Const_4000_Hex) OTE(MCC2_15E_CommsOK) ,E300ToMotor(AOI_MCC2_15E_ToPLC1,MotorsStatusTag.MCC2_15E,AOP_MCC2_15E:I,MCC2_15E_CommsOK) ];
   71: [GSV(Module,AOP_MCC2_15G,EntryStatus,GSV_EntryStatus) MEQ(GSV_EntryStatus,16#f000,Const_4000_Hex) OTE(MCC2_15G_CommsOK) ,E300ToMotor(AOI_MCC2_15G_ToPLC1,MotorsStatusTag.MCC2_15G,AOP_MCC2_15G:I,MCC2_15G_CommsOK) ];
